{attribute 'qualified_only'} // Variable needs to be used with ENUM name
{attribute 'strict'} // Strict rules, prevents invalid assignments/mathematical operations on the ENUM

TYPE E_Mode : // List of settings the program can use, different modes
(
	Off := 0,
	Auto := 1,
	Manuel := 2
);
END_TYPE

(* stored: Version 1.1.0.1
   DUT E_Mode: Id {e8599410-a039-46f7-81be-1321c5e77880} *)
